TYPE ST_KPI_CodePos :
STRUCT
	ReadOK				: UDINT;
	Efficiency			: LREAL;
END_STRUCT
END_TYPE

(* stored: Version 1.1.0.1, ProductVersion 3.1.4024.15
   DUT ST_KPI_CodePos: Id {96de2758-6652-4c2c-bf7b-df424230f0cc} *)
